// TIA Portal V17 export
// export: Created 2025-03-05T08:00:02.6959975Z, ExportSetting WithDefaults, DisplayName Totally Integrated Automation Portal, DisplayVersion V17 Update 8, DisplayName TIA Portal Openness, DisplayVersion V17 Update 8, DisplayName TIA Portal Version Control Interface, DisplayVersion V17, DisplayName SINAMICS Startdrive Advanced, DisplayVersion V17 SP2, DisplayName SINAMICS Startdrive G110M, G120, G120C, G120D, G120P, G115D, DisplayVersion V17 SP2, DisplayName SINAMICS Startdrive G130, G150, S120, S150, SINAMICS MV, S210, DisplayVersion V17 SP2, DisplayName STEP 7 Professional, DisplayVersion V17 Update 8, DisplayName SINUMERIK ONE STEP 7 Toolbox, DisplayVersion V17 Update 12, DisplayName SINUMERIK 840D sl STEP 7 Toolbox, DisplayVersion V17 Update 12, DisplayName STEP 7 Safety, DisplayVersion V17 Update 6, DisplayName WinCC Advanced, DisplayVersion V17 Update 8
FUNCTION "FC2003_CNC_MODES_G1" : Void   // FC2003, LAD
{ S7_Optimized_Access := 'FALSE' }
AUTHOR : ETXETAR
VERSION : 1.0
// stored: AutoNumber false, IsIECCheckEnabled false, SetENOAutomatically false, UDAEnableTagReadback false
   VAR CONSTANT
      FC_NUMBER : DInt := 2003;
   END_VAR
BEGIN

NETWORK
TITLE = ACTUAL VALUE IN WCS 0=MCS / Actual value in WCS 0=MCS
// WKS/MKS
      AN    "LBP_HMI".E_ActWCS;
      JC    M001;
      AN    "LBP_HMI".A_ActWCS;
      =     "LBP_HMI".A_ActWCS;
      CLR;
      =     "LBP_HMI".E_ActWCS;
M001: NOP   0;

REGION Network 2: MODE GROUP RESET / Mode group reset
   // BAG Reset
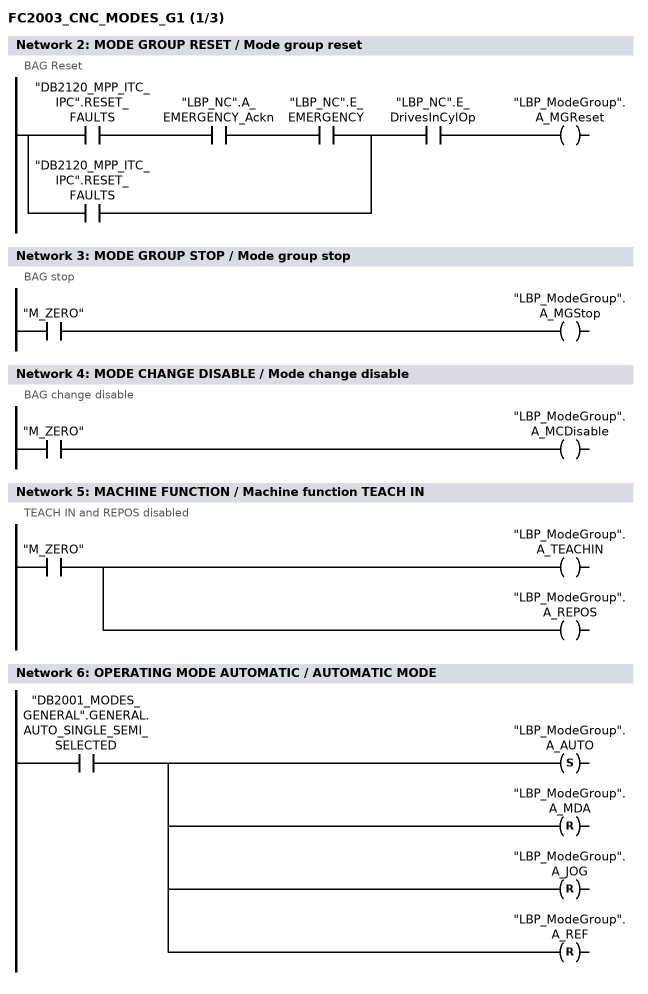
   RUNG wire#powerrail
      Contact( "DB2120_MPP_ITC_IPC".RESET_FAULTS )
      Contact( "LBP_NC".A_EMERGENCY_Ackn )
      Contact( "LBP_NC".E_EMERGENCY )
      wire#w1
      Contact( "LBP_NC".E_DrivesInCylOp )
      Coil( "LBP_ModeGroup".A_MGReset )
   END_RUNG
   RUNG wire#powerrail
      Contact( "DB2120_MPP_ITC_IPC".RESET_FAULTS )
   END_RUNG wire#w1
   // the same network as SCL:
   "LBP_ModeGroup".A_MGReset := (("DB2120_MPP_ITC_IPC".RESET_FAULTS AND "LBP_NC".A_EMERGENCY_Ackn AND "LBP_NC".E_EMERGENCY) OR "DB2120_MPP_ITC_IPC".RESET_FAULTS) AND "LBP_NC".E_DrivesInCylOp;
END_REGION

REGION Network 3: MODE GROUP STOP / Mode group stop
   // BAG stop
   RUNG wire#powerrail
      Contact( "M_ZERO" )
      Coil( "LBP_ModeGroup".A_MGStop )
   END_RUNG
   // the same network as SCL:
   "LBP_ModeGroup".A_MGStop := "M_ZERO";
END_REGION

REGION Network 4: MODE CHANGE DISABLE / Mode change disable
   // BAG change disable
   RUNG wire#powerrail
      Contact( "M_ZERO" )
      Coil( "LBP_ModeGroup".A_MCDisable )
   END_RUNG
   // the same network as SCL:
   "LBP_ModeGroup".A_MCDisable := "M_ZERO";
END_REGION

REGION Network 5: MACHINE FUNCTION / Machine function TEACH IN
   // TEACH IN and REPOS disabled
   RUNG wire#powerrail
      Contact( "M_ZERO" )
      wire#w1
      Coil( "LBP_ModeGroup".A_TEACHIN )
   END_RUNG
   RUNG wire#w1
      Coil( "LBP_ModeGroup".A_REPOS )
   END_RUNG
   // the same network as SCL:
   "LBP_ModeGroup".A_TEACHIN := "M_ZERO";
   "LBP_ModeGroup".A_REPOS := "M_ZERO";
END_REGION

REGION Network 6: OPERATING MODE AUTOMATIC / AUTOMATIC MODE
   RUNG wire#powerrail
      Contact( "DB2001_MODES_GENERAL".GENERAL.AUTO_SINGLE_SEMI_SELECTED )
      wire#w1
      S_Coil( "LBP_ModeGroup".A_AUTO )
   END_RUNG
   RUNG wire#w1
      R_Coil( "LBP_ModeGroup".A_MDA )
   END_RUNG
   RUNG wire#w1
      R_Coil( "LBP_ModeGroup".A_JOG )
   END_RUNG
   RUNG wire#w1
      R_Coil( "LBP_ModeGroup".A_REF )
   END_RUNG
   // the same network as SCL:
   IF "DB2001_MODES_GENERAL".GENERAL.AUTO_SINGLE_SEMI_SELECTED THEN
       "LBP_ModeGroup".A_AUTO := TRUE;
       "LBP_ModeGroup".A_MDA := FALSE;
       "LBP_ModeGroup".A_JOG := FALSE;
       "LBP_ModeGroup".A_REF := FALSE;
   END_IF;
END_REGION

REGION Network 7: OPERATING MODE MDA / MDI MODE
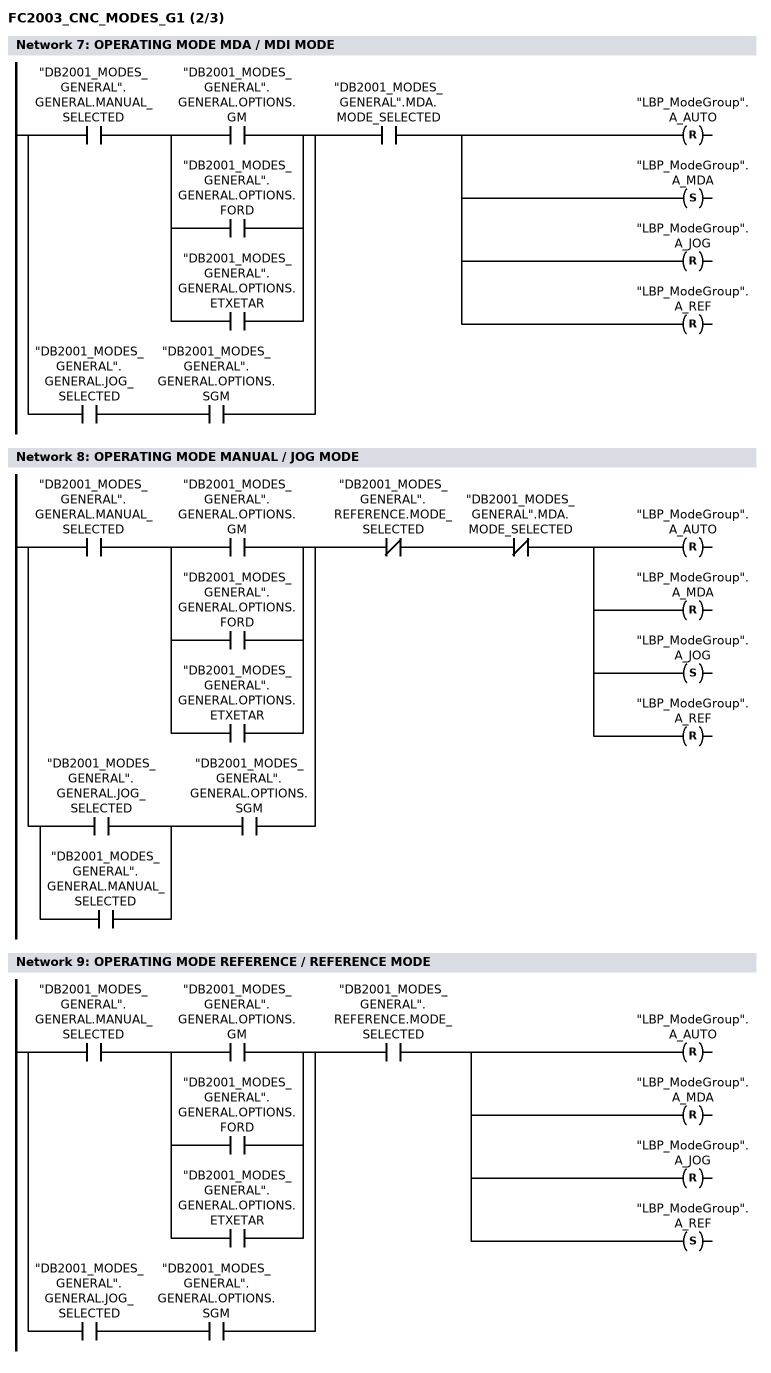
   RUNG wire#powerrail
      Contact( "DB2001_MODES_GENERAL".GENERAL.MANUAL_SELECTED )
      wire#w1
      Contact( "DB2001_MODES_GENERAL".GENERAL.OPTIONS.GM )
      wire#w2
      Contact( "DB2001_MODES_GENERAL".MDA.MODE_SELECTED )
      wire#w3
      R_Coil( "LBP_ModeGroup".A_AUTO )
   END_RUNG
   RUNG wire#w1
      Contact( "DB2001_MODES_GENERAL".GENERAL.OPTIONS.FORD )
   END_RUNG wire#w2
   RUNG wire#w1
      Contact( "DB2001_MODES_GENERAL".GENERAL.OPTIONS.ETXETAR )
   END_RUNG wire#w2
   RUNG wire#powerrail
      Contact( "DB2001_MODES_GENERAL".GENERAL.JOG_SELECTED )
      Contact( "DB2001_MODES_GENERAL".GENERAL.OPTIONS.SGM )
   END_RUNG wire#w2
   RUNG wire#w3
      S_Coil( "LBP_ModeGroup".A_MDA )
   END_RUNG
   RUNG wire#w3
      R_Coil( "LBP_ModeGroup".A_JOG )
   END_RUNG
   RUNG wire#w3
      R_Coil( "LBP_ModeGroup".A_REF )
   END_RUNG
   // the same network as SCL:
   IF (("DB2001_MODES_GENERAL".GENERAL.MANUAL_SELECTED AND ("DB2001_MODES_GENERAL".GENERAL.OPTIONS.GM OR "DB2001_MODES_GENERAL".GENERAL.OPTIONS.FORD OR "DB2001_MODES_GENERAL".GENERAL.OPTIONS.ETXETAR)) OR ("DB2001_MODES_GENERAL".GENERAL.JOG_SELECTED AND "DB2001_MODES_GENERAL".GENERAL.OPTIONS.SGM)) AND "DB2001_MODES_GENERAL".MDA.MODE_SELECTED THEN
       "LBP_ModeGroup".A_AUTO := FALSE;
       "LBP_ModeGroup".A_MDA := TRUE;
       "LBP_ModeGroup".A_JOG := FALSE;
       "LBP_ModeGroup".A_REF := FALSE;
   END_IF;
END_REGION

REGION Network 8: OPERATING MODE MANUAL / JOG MODE
   RUNG wire#powerrail
      Contact( "DB2001_MODES_GENERAL".GENERAL.MANUAL_SELECTED )
      wire#w1
      Contact( "DB2001_MODES_GENERAL".GENERAL.OPTIONS.GM )
      wire#w2
      I_Contact( "DB2001_MODES_GENERAL".REFERENCE.MODE_SELECTED )
      I_Contact( "DB2001_MODES_GENERAL".MDA.MODE_SELECTED )
      wire#w4
      R_Coil( "LBP_ModeGroup".A_AUTO )
   END_RUNG
   RUNG wire#w1
      Contact( "DB2001_MODES_GENERAL".GENERAL.OPTIONS.FORD )
   END_RUNG wire#w2
   RUNG wire#w1
      Contact( "DB2001_MODES_GENERAL".GENERAL.OPTIONS.ETXETAR )
   END_RUNG wire#w2
   RUNG wire#powerrail
      Contact( "DB2001_MODES_GENERAL".GENERAL.JOG_SELECTED )
      wire#w3
      Contact( "DB2001_MODES_GENERAL".GENERAL.OPTIONS.SGM )
   END_RUNG wire#w2
   RUNG wire#powerrail
      Contact( "DB2001_MODES_GENERAL".GENERAL.MANUAL_SELECTED )
   END_RUNG wire#w3
   RUNG wire#w4
      R_Coil( "LBP_ModeGroup".A_MDA )
   END_RUNG
   RUNG wire#w4
      S_Coil( "LBP_ModeGroup".A_JOG )
   END_RUNG
   RUNG wire#w4
      R_Coil( "LBP_ModeGroup".A_REF )
   END_RUNG
   // the same network as SCL:
   IF (("DB2001_MODES_GENERAL".GENERAL.MANUAL_SELECTED AND ("DB2001_MODES_GENERAL".GENERAL.OPTIONS.GM OR "DB2001_MODES_GENERAL".GENERAL.OPTIONS.FORD OR "DB2001_MODES_GENERAL".GENERAL.OPTIONS.ETXETAR)) OR (("DB2001_MODES_GENERAL".GENERAL.JOG_SELECTED OR "DB2001_MODES_GENERAL".GENERAL.MANUAL_SELECTED) AND "DB2001_MODES_GENERAL".GENERAL.OPTIONS.SGM)) AND NOT "DB2001_MODES_GENERAL".REFERENCE.MODE_SELECTED AND NOT "DB2001_MODES_GENERAL".MDA.MODE_SELECTED THEN
       "LBP_ModeGroup".A_AUTO := FALSE;
       "LBP_ModeGroup".A_MDA := FALSE;
       "LBP_ModeGroup".A_JOG := TRUE;
       "LBP_ModeGroup".A_REF := FALSE;
   END_IF;
END_REGION

REGION Network 9: OPERATING MODE REFERENCE / REFERENCE MODE
   RUNG wire#powerrail
      Contact( "DB2001_MODES_GENERAL".GENERAL.MANUAL_SELECTED )
      wire#w1
      Contact( "DB2001_MODES_GENERAL".GENERAL.OPTIONS.GM )
      wire#w2
      Contact( "DB2001_MODES_GENERAL".REFERENCE.MODE_SELECTED )
      wire#w3
      R_Coil( "LBP_ModeGroup".A_AUTO )
   END_RUNG
   RUNG wire#w1
      Contact( "DB2001_MODES_GENERAL".GENERAL.OPTIONS.FORD )
   END_RUNG wire#w2
   RUNG wire#w1
      Contact( "DB2001_MODES_GENERAL".GENERAL.OPTIONS.ETXETAR )
   END_RUNG wire#w2
   RUNG wire#powerrail
      Contact( "DB2001_MODES_GENERAL".GENERAL.JOG_SELECTED )
      Contact( "DB2001_MODES_GENERAL".GENERAL.OPTIONS.SGM )
   END_RUNG wire#w2
   RUNG wire#w3
      R_Coil( "LBP_ModeGroup".A_MDA )
   END_RUNG
   RUNG wire#w3
      R_Coil( "LBP_ModeGroup".A_JOG )
   END_RUNG
   RUNG wire#w3
      S_Coil( "LBP_ModeGroup".A_REF )
   END_RUNG
   // the same network as SCL:
   IF (("DB2001_MODES_GENERAL".GENERAL.MANUAL_SELECTED AND ("DB2001_MODES_GENERAL".GENERAL.OPTIONS.GM OR "DB2001_MODES_GENERAL".GENERAL.OPTIONS.FORD OR "DB2001_MODES_GENERAL".GENERAL.OPTIONS.ETXETAR)) OR ("DB2001_MODES_GENERAL".GENERAL.JOG_SELECTED AND "DB2001_MODES_GENERAL".GENERAL.OPTIONS.SGM)) AND "DB2001_MODES_GENERAL".REFERENCE.MODE_SELECTED THEN
       "LBP_ModeGroup".A_AUTO := FALSE;
       "LBP_ModeGroup".A_MDA := FALSE;
       "LBP_ModeGroup".A_JOG := FALSE;
       "LBP_ModeGroup".A_REF := TRUE;
   END_IF;
END_REGION

REGION Network 10: OPERATING MODE NO MODE / NO REFERENCE MODE
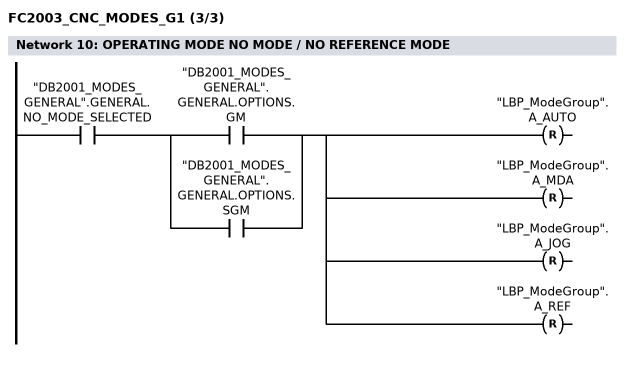
   RUNG wire#powerrail
      Contact( "DB2001_MODES_GENERAL".GENERAL.NO_MODE_SELECTED )
      wire#w1
      Contact( "DB2001_MODES_GENERAL".GENERAL.OPTIONS.GM )
      wire#w2
      R_Coil( "LBP_ModeGroup".A_AUTO )
   END_RUNG
   RUNG wire#w1
      Contact( "DB2001_MODES_GENERAL".GENERAL.OPTIONS.SGM )
   END_RUNG wire#w2
   RUNG wire#w2
      R_Coil( "LBP_ModeGroup".A_MDA )
   END_RUNG
   RUNG wire#w2
      R_Coil( "LBP_ModeGroup".A_JOG )
   END_RUNG
   RUNG wire#w2
      R_Coil( "LBP_ModeGroup".A_REF )
   END_RUNG
   // the same network as SCL:
   IF "DB2001_MODES_GENERAL".GENERAL.NO_MODE_SELECTED AND ("DB2001_MODES_GENERAL".GENERAL.OPTIONS.GM OR "DB2001_MODES_GENERAL".GENERAL.OPTIONS.SGM) THEN
       "LBP_ModeGroup".A_AUTO := FALSE;
       "LBP_ModeGroup".A_MDA := FALSE;
       "LBP_ModeGroup".A_JOG := FALSE;
       "LBP_ModeGroup".A_REF := FALSE;
   END_IF;
END_REGION
END_FUNCTION
